FUNCTION_BLOCK FB_DiagnosisEtherCATSlaveWc0
VAR_OUTPUT
	bError						:BOOL;								//エラー発生を出力
END_VAR
VAR
	fbStateDiagnosis			:FB_StateDiagnosis;
END_VAR

//診断用FBを呼び出し
fbStateDiagnosis();

bError:=fbStateDiagnosis.bError;

END_FUNCTION_BLOCK

(* stored: Version 1.1.0.1, ProductVersion 3.1.4026.18
   POU FB_DiagnosisEtherCATSlaveWc0: Id {519e11a6-b44d-418f-ae09-7534acbef856}, SpecialFunc None *)
